{attribute 'linkalways'} 
{attribute 'no_explicit_call' := 'This FB is a CLASS and must be accessed using methods or properties'}
{attribute 'enable_dynamic_creation'}
FUNCTION_BLOCK FINAL ADD_ULINT EXTENDS Node
VAR
	in1 : _ULINT(0);
	in2 : _ULINT(0);
	out : _ULINT(0);
END_VAR

METHOD PUBLIC Clone : I_Node
VAR
	pNode : POINTER TO ADD_ULINT;
END_VAR
pNode := __NEW(ADD_ULINT);
Clone := pNode^;
END_METHOD

METHOD FB_init : BOOL
VAR_INPUT
	bInitRetains : BOOL; // if TRUE, the retain variables are initialized (warm start / cold start)
	bInCopyCode : BOOL;  // if TRUE, the instance afterwards gets moved into the copy code (online change)
END_VAR
AddInput('in1',THIS^.in1);
AddInput('in2',THIS^.in2);
AddOutput('out', THIS^.out);
END_METHOD

METHOD PROTECTED OnExecute
VAR
END_VAR
out.Value := in1.Value + in2.Value;
END_METHOD

END_FUNCTION_BLOCK

(* stored: Version 1.1.0.1, ProductVersion 3.1.4024.15
   POU ADD_ULINT: Id {61240e48-b59c-4f35-a44e-3f9a5e969ab0}, SpecialFunc None
   Folder Constructor: Id {0507fc12-b9e8-4ada-a480-4ae23a7649d5}
   Method Clone: Id {88854625-7e34-4fbc-bb7a-c5b95e76389b}
   Method FB_init: Id {6e1975e8-955f-49d3-ab8a-fa85f9e7f7b6}
   Method OnExecute: Id {8ce62cb4-49ec-4d73-93d8-ba9be7922f2d} *)
